(* PLC project Unnamed, Unknown Unnamed 1 *)
(* stored: creationDateTime 2023-02-06T11:08:00, modificationDateTime 2023-02-07T21:25:46 *)

PROGRAM program0
  VAR CONSTANT
    always_true : BOOL := 1;
    always_false : BOOL := 0;
  END_VAR
  VAR
    moving_x AT %IX100.0 : BOOL;
    moving_z AT %IX100.1 : BOOL;
    item_detected AT %IX100.2 : BOOL;
    lid_at_place AT %IX100.3 : BOOL;
    lid_clamped AT %IX100.4 : BOOL;
    pos_at_limit_lid AT %IX100.5 : BOOL;
    base_at_place AT %IX100.6 : BOOL;
    base_clamped AT %IX100.7 : BOOL;
    pos_at_limit_base AT %IX101.0 : BOOL;
    part_leaving AT %IX101.1 : BOOL;
    start AT %IX101.2 : BOOL;
    reset AT %IX101.3 : BOOL;
    stop AT %IX101.4 : BOOL;
    estop AT %IX101.5 : BOOL;
    auto AT %IX101.6 : BOOL;
    factoryio_running AT %IX101.7 : BOOL;
    move_x AT %QX100.0 : BOOL;
    move_z AT %QX100.1 : BOOL;
    grab AT %QX100.2 : BOOL;
    lids_conveyor AT %QX100.3 : BOOL;
    clamp_lid AT %QX100.4 : BOOL;
    pos_raise_lid AT %QX100.5 : BOOL;
    bases_conveyor AT %QX100.6 : BOOL;
    clamp_base AT %QX100.7 : BOOL;
    pos_raise_base AT %QX101.0 : BOOL;
    bases_emitter AT %QX101.1 : BOOL;
    lids_emitter AT %QX101.2 : BOOL;
    stop_light AT %QX101.3 : BOOL;
  END_VAR
  VAR
    machine_ready : BOOL;
    start_emitters : BOOL;
    emit_next : BOOL;
    process_started : BOOL;
    process_finished : BOOL;
    step_num : INT;
    first_part : BOOL;
    base_ready : BOOL;
    lid_ready : BOOL;
    F_TRIG0 : F_TRIG;
    F_TRIG1 : F_TRIG;
    TON0 : TON;
  END_VAR

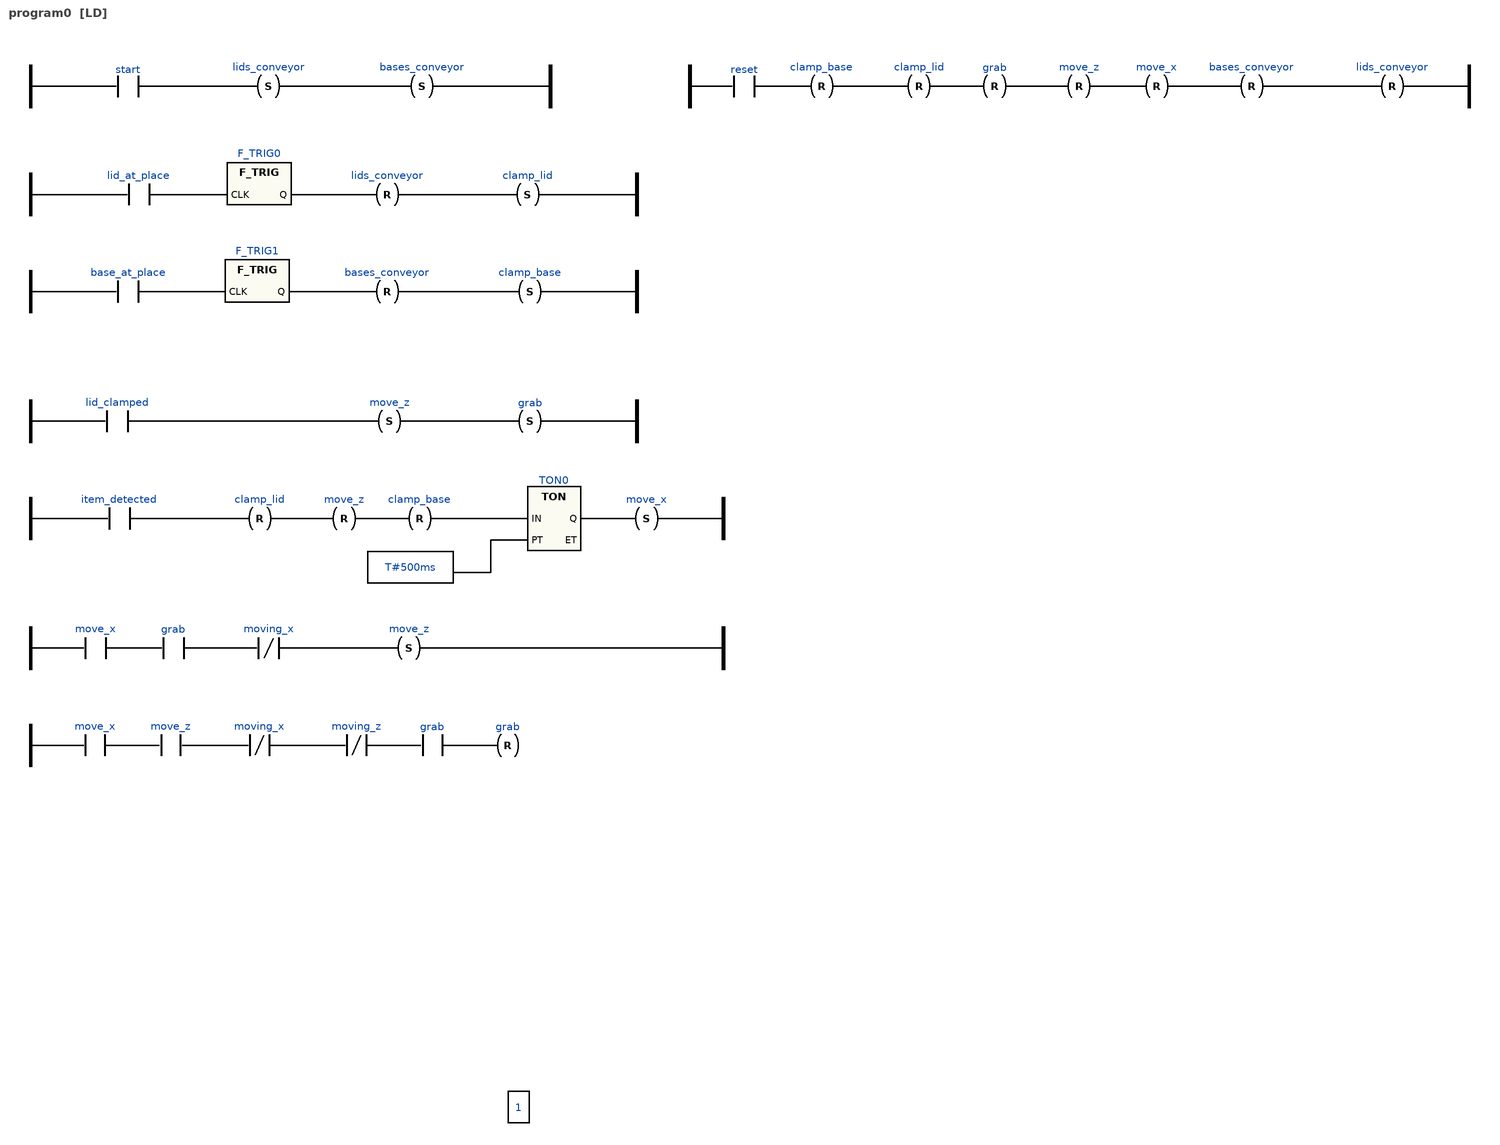
(* LD diagram, written out as Structured Text *)
IF start THEN lids_conveyor := TRUE; END_IF;
IF start THEN bases_conveyor := TRUE; END_IF;
IF reset THEN clamp_base := FALSE; END_IF;
IF reset THEN clamp_lid := FALSE; END_IF;
IF reset THEN grab := FALSE; END_IF;
IF reset THEN move_z := FALSE; END_IF;
IF reset THEN move_x := FALSE; END_IF;
IF reset THEN bases_conveyor := FALSE; END_IF;
IF reset THEN lids_conveyor := FALSE; END_IF;
F_TRIG0(CLK := lid_at_place);
IF F_TRIG0.Q THEN lids_conveyor := FALSE; END_IF;
IF F_TRIG0.Q THEN clamp_lid := TRUE; END_IF;
F_TRIG1(CLK := base_at_place);
IF F_TRIG1.Q THEN bases_conveyor := FALSE; END_IF;
IF F_TRIG1.Q THEN clamp_base := TRUE; END_IF;
IF lid_clamped THEN move_z := TRUE; END_IF;
IF lid_clamped THEN grab := TRUE; END_IF;
IF item_detected THEN clamp_lid := FALSE; END_IF;
IF item_detected THEN move_z := FALSE; END_IF;
IF item_detected THEN clamp_base := FALSE; END_IF;
TON0(IN := item_detected, PT := T#500ms);
IF TON0.Q THEN move_x := TRUE; END_IF;
IF move_x AND grab AND NOT moving_x THEN move_z := TRUE; END_IF;
IF move_x AND move_z AND NOT moving_x AND NOT moving_z AND grab THEN grab := FALSE; END_IF;
(* drawn but not wired to any output: 1 *)
END_PROGRAM

CONFIGURATION Config0
  RESOURCE Res0 ON PLC
    TASK task0(INTERVAL := T#20ms, PRIORITY := 0);
    PROGRAM instance0 WITH task0 : program0;
  END_RESOURCE
END_CONFIGURATION
